{attribute addProperty BoxType "EPP2339-0003-0016"}
{attribute addProperty Id "OutputAT %Q*ARRAY[0 ..7] OF BOOL6480"}
{attribute addProperty CRC "1062725746"}
{attribute addProperty SizeInBites "64"}
{attribute addProperty SizeInBytes "8"}
TYPE DO_Outputs_Channel_33B76376 :
STRUCT
	{attribute addProperty Name "Output"}
	Output AT %Q* : ARRAY[0 ..7] OF BOOL;
END_STRUCT
END_TYPE

(* stored: Version 1.2.0.0, ProductVersion 3.1.4024.9
   DUT DO_Outputs_Channel_33B76376: Id {71997797-4443-4cd0-978f-0d854134ed78} *)
